            Abre_Comp_Indiv_Gar_1 = FALSE
            Fecha_Comp_Indiv_Gar_1 = TRUE

            Abre_Comp_Indiv_Gar_3 = FALSE
            Fecha_Comp_Indiv_Gar_3 = TRUE

            Abre_Comp_Indiv_Gar_4 = FALSE
            Fecha_Comp_Indiv_Gar_4 = TRUE

            Abre_Comp_Indiv_Gar_6 = FALSE
            Fecha_Comp_Indiv_Gar_6 = TRUE

            Ava_Cil_1_Gar_1 = TRUE
            Rec_Cil_1_Gar_1 = FALSE

            Ava_Cil_1_Gar_2 = TRUE
            Rec_Cil_1_Gar_2 = FALSE

            Ava_Cil_1_Gar_3 = TRUE
            Rec_Cil_1_Gar_3 = FALSE

            Ava_Cil_1_Gar_4 = TRUE
            Rec_Cil_1_Gar_4 = FALSE

            Ava_Cil_1_Gar_5 = TRUE
            Rec_Cil_1_Gar_5 = FALSE

            Ava_Cil_1_Gar_6 = TRUE
            Rec_Cil_1_Gar_6 = FALSE

            Ava_Cil_2_Gar_1 = TRUE
            Rec_Cil_2_Gar_1 = FALSE

            Ava_Cil_2_Gar_2 = TRUE
            Rec_Cil_2_Gar_2 = FALSE

            Ava_Cil_2_Gar_3 = TRUE
            Rec_Cil_2_Gar_3 = FALSE

            Ava_Cil_2_Gar_4 = TRUE
            Rec_Cil_2_Gar_4 = FALSE

            Ava_Cil_2_Gar_5 = TRUE
            Rec_Cil_2_Gar_5 = FALSE

            Ava_Cil_2_Gar_6 = TRUE
            Rec_Cil_2_Gar_6 = FALSE



         CASE 162
            Abre_Gar_Triplo_Lado_A = TRUE
            Fecha_Gar_Triplo_Lado_A = FALSE

            Abre_Gar_Triplo_Lado_B = TRUE
            Fecha_Gar_Triplo_Lado_B = FALSE

            Abre_Comp_Indiv_Gar_1 = FALSE
            Fecha_Comp_Indiv_Gar_1 = TRUE

            Abre_Comp_Indiv_Gar_3 = FALSE
            Fecha_Comp_Indiv_Gar_3 = TRUE

            Abre_Comp_Indiv_Gar_4 = FALSE
            Fecha_Comp_Indiv_Gar_4 = TRUE

            Abre_Comp_Indiv_Gar_6 = TRUE
            Fecha_Comp_Indiv_Gar_6 = FALSE

            Ava_Cil_1_Gar_1 = TRUE
            Rec_Cil_1_Gar_1 = FALSE

            Ava_Cil_1_Gar_2 = TRUE
            Rec_Cil_1_Gar_2 = FALSE

            Ava_Cil_1_Gar_3 = TRUE
            Rec_Cil_1_Gar_3 = FALSE

            Ava_Cil_1_Gar_4 = TRUE
            Rec_Cil_1_Gar_4 = FALSE

            Ava_Cil_1_Gar_5 = TRUE
            Rec_Cil_1_Gar_5 = FALSE

            Ava_Cil_1_Gar_6 = TRUE
            Rec_Cil_1_Gar_6 = FALSE

            Ava_Cil_2_Gar_1 = TRUE
            Rec_Cil_2_Gar_1 = FALSE

            Ava_Cil_2_Gar_2 = TRUE
            Rec_Cil_2_Gar_2 = FALSE

            Ava_Cil_2_Gar_3 = TRUE
            Rec_Cil_2_Gar_3 = FALSE

            Ava_Cil_2_Gar_4 = TRUE
            Rec_Cil_2_Gar_4 = FALSE

            Ava_Cil_2_Gar_5 = TRUE
            Rec_Cil_2_Gar_5 = FALSE

            Ava_Cil_2_Gar_6 = TRUE
            Rec_Cil_2_Gar_6 = FALSE

         CASE 61
            Abre_Gar_Triplo_Lado_A = TRUE
            Fecha_Gar_Triplo_Lado_A = FALSE

            Abre_Gar_Triplo_Lado_B = TRUE
            Fecha_Gar_Triplo_Lado_B = FALSE

            Abre_Comp_Indiv_Gar_1 = TRUE
            Fecha_Comp_Indiv_Gar_1 = FALSE

            Abre_Comp_Indiv_Gar_3 = FALSE
            Fecha_Comp_Indiv_Gar_3 = TRUE

            Abre_Comp_Indiv_Gar_4 = FALSE
            Fecha_Comp_Indiv_Gar_4 = TRUE

            Abre_Comp_Indiv_Gar_6 = TRUE
            Fecha_Comp_Indiv_Gar_6 = FALSE

            Ava_Cil_1_Gar_1 = TRUE
            Rec_Cil_1_Gar_1 = FALSE

            Ava_Cil_1_Gar_2 = TRUE
            Rec_Cil_1_Gar_2 = FALSE

            Ava_Cil_1_Gar_3 = TRUE
            Rec_Cil_1_Gar_3 = FALSE

            Ava_Cil_1_Gar_4 = TRUE
            Rec_Cil_1_Gar_4 = FALSE

            Ava_Cil_1_Gar_5 = TRUE
            Rec_Cil_1_Gar_5 = FALSE

            Ava_Cil_1_Gar_6 = TRUE
            Rec_Cil_1_Gar_6 = FALSE

            Ava_Cil_2_Gar_1 = TRUE
            Rec_Cil_2_Gar_1 = FALSE

            Ava_Cil_2_Gar_2 = TRUE
            Rec_Cil_2_Gar_2 = FALSE

            Ava_Cil_2_Gar_3 = TRUE
            Rec_Cil_2_Gar_3 = FALSE

            Ava_Cil_2_Gar_4 = TRUE
            Rec_Cil_2_Gar_4 = FALSE

            Ava_Cil_2_Gar_5 = TRUE
            Rec_Cil_2_Gar_5 = FALSE

            Ava_Cil_2_Gar_6 = TRUE
            Rec_Cil_2_Gar_6 = FALSE


         CASE 62
            Abre_Gar_Triplo_Lado_A = TRUE
            Fecha_Gar_Triplo_Lado_A = FALSE

            Abre_Gar_Triplo_Lado_B = TRUE
            Fecha_Gar_Triplo_Lado_B = FALSE

            Abre_Comp_Indiv_Gar_1 = TRUE
            Fecha_Comp_Indiv_Gar_1 = FALSE

            Abre_Comp_Indiv_Gar_3 = FALSE
            Fecha_Comp_Indiv_Gar_3 = TRUE

            Abre_Comp_Indiv_Gar_4 = FALSE
            Fecha_Comp_Indiv_Gar_4 = TRUE

            Abre_Comp_Indiv_Gar_6 = TRUE
            Fecha_Comp_Indiv_Gar_6 = FALSE

            Ava_Cil_1_Gar_1 = TRUE
            Rec_Cil_1_Gar_1 = FALSE

            Ava_Cil_1_Gar_2 = TRUE
            Rec_Cil_1_Gar_2 = FALSE

            Ava_Cil_1_Gar_3 = TRUE
            Rec_Cil_1_Gar_3 = FALSE

            Ava_Cil_1_Gar_4 = TRUE
            Rec_Cil_1_Gar_4 = FALSE

            Ava_Cil_1_Gar_5 = TRUE
            Rec_Cil_1_Gar_5 = FALSE

            Ava_Cil_1_Gar_6 = TRUE
            Rec_Cil_1_Gar_6 = FALSE

            Ava_Cil_2_Gar_1 = TRUE
            Rec_Cil_2_Gar_1 = FALSE

            Ava_Cil_2_Gar_2 = TRUE
            Rec_Cil_2_Gar_2 = FALSE

            Ava_Cil_2_Gar_3 = TRUE
            Rec_Cil_2_Gar_3 = FALSE

            Ava_Cil_2_Gar_4 = TRUE
            Rec_Cil_2_Gar_4 = FALSE

            Ava_Cil_2_Gar_5 = TRUE
            Rec_Cil_2_Gar_5 = FALSE

            Ava_Cil_2_Gar_6 = TRUE
            Rec_Cil_2_Gar_6 = FALSE

         CASE 191
            Abre_Gar_Triplo_Lado_A = TRUE
            Fecha_Gar_Triplo_Lado_A = FALSE

            Abre_Gar_Triplo_Lado_B = TRUE
            Fecha_Gar_Triplo_Lado_B = FALSE

            Abre_Comp_Indiv_Gar_1 = FALSE
            Fecha_Comp_Indiv_Gar_1 = TRUE

            Abre_Comp_Indiv_Gar_3 = FALSE
            Fecha_Comp_Indiv_Gar_3 = TRUE

            Abre_Comp_Indiv_Gar_4 = FALSE
            Fecha_Comp_Indiv_Gar_4 = TRUE

            Abre_Comp_Indiv_Gar_6 = FALSE
            Fecha_Comp_Indiv_Gar_6 = TRUE

            Ava_Cil_1_Gar_1 = TRUE
            Rec_Cil_1_Gar_1 = FALSE

            Ava_Cil_1_Gar_2 = TRUE
            Rec_Cil_1_Gar_2 = FALSE

            Ava_Cil_1_Gar_3 = TRUE
            Rec_Cil_1_Gar_3 = FALSE

            Ava_Cil_1_Gar_4 = TRUE
            Rec_Cil_1_Gar_4 = FALSE

            Ava_Cil_1_Gar_5 = TRUE
            Rec_Cil_1_Gar_5 = FALSE

            Ava_Cil_1_Gar_6 = TRUE
            Rec_Cil_1_Gar_6 = FALSE

            Ava_Cil_2_Gar_1 = TRUE
            Rec_Cil_2_Gar_1 = FALSE

            Ava_Cil_2_Gar_2 = TRUE
            Rec_Cil_2_Gar_2 = FALSE

            Ava_Cil_2_Gar_3 = TRUE
            Rec_Cil_2_Gar_3 = FALSE

            Ava_Cil_2_Gar_4 = TRUE
            Rec_Cil_2_Gar_4 = FALSE

            Ava_Cil_2_Gar_5 = TRUE
            Rec_Cil_2_Gar_5 = FALSE

            Ava_Cil_2_Gar_6 = TRUE
            Rec_Cil_2_Gar_6 = FALSE

         CASE 192
            Abre_Gar_Triplo_Lado_A = TRUE
            Fecha_Gar_Triplo_Lado_A = FALSE

            Abre_Gar_Triplo_Lado_B = TRUE
            Fecha_Gar_Triplo_Lado_B = FALSE

            Abre_Comp_Indiv_Gar_1 = FALSE
            Fecha_Comp_Indiv_Gar_1 = TRUE

            Abre_Comp_Indiv_Gar_3 = FALSE
            Fecha_Comp_Indiv_Gar_3 = TRUE

            Abre_Comp_Indiv_Gar_4 = FALSE
            Fecha_Comp_Indiv_Gar_4 = TRUE

            Abre_Comp_Indiv_Gar_6 = FALSE
            Fecha_Comp_Indiv_Gar_6 = TRUE

            Ava_Cil_1_Gar_1 = TRUE
            Rec_Cil_1_Gar_1 = FALSE

            Ava_Cil_1_Gar_2 = TRUE
            Rec_Cil_1_Gar_2 = FALSE

            Ava_Cil_1_Gar_3 = TRUE
            Rec_Cil_1_Gar_3 = FALSE

            Ava_Cil_1_Gar_4 = TRUE
            Rec_Cil_1_Gar_4 = FALSE

            Ava_Cil_1_Gar_5 = TRUE
            Rec_Cil_1_Gar_5 = FALSE

            Ava_Cil_1_Gar_6 = TRUE
            Rec_Cil_1_Gar_6 = FALSE

            Ava_Cil_2_Gar_1 = TRUE
            Rec_Cil_2_Gar_1 = FALSE

            Ava_Cil_2_Gar_2 = TRUE
            Rec_Cil_2_Gar_2 = FALSE

            Ava_Cil_2_Gar_3 = TRUE
            Rec_Cil_2_Gar_3 = FALSE

            Ava_Cil_2_Gar_4 = TRUE
            Rec_Cil_2_Gar_4 = FALSE

            Ava_Cil_2_Gar_5 = TRUE
            Rec_Cil_2_Gar_5 = FALSE

            Ava_Cil_2_Gar_6 = TRUE
            Rec_Cil_2_Gar_6 = FALSE

         CASE 81
            Abre_Gar_Triplo_Lado_A = TRUE
            Fecha_Gar_Triplo_Lado_A = FALSE

            Abre_Gar_Triplo_Lado_B = TRUE
            Fecha_Gar_Triplo_Lado_B = FALSE

            Abre_Comp_Indiv_Gar_1 = FALSE
            Fecha_Comp_Indiv_Gar_1 = TRUE

            Abre_Comp_Indiv_Gar_3 = FALSE
            Fecha_Comp_Indiv_Gar_3 = TRUE

            Abre_Comp_Indiv_Gar_4 = FALSE
            Fecha_Comp_Indiv_Gar_4 = TRUE

            Abre_Comp_Indiv_Gar_6 = TRUE
            Fecha_Comp_Indiv_Gar_6 = FALSE

            Ava_Cil_1_Gar_1 = TRUE
            Rec_Cil_1_Gar_1 = FALSE

            Ava_Cil_1_Gar_2 = TRUE
            Rec_Cil_1_Gar_2 = FALSE

            Ava_Cil_1_Gar_3 = TRUE
            Rec_Cil_1_Gar_3 = FALSE

            Ava_Cil_1_Gar_4 = TRUE
            Rec_Cil_1_Gar_4 = FALSE

            Ava_Cil_1_Gar_5 = TRUE
            Rec_Cil_1_Gar_5 = FALSE

            Ava_Cil_1_Gar_6 = TRUE
            Rec_Cil_1_Gar_6 = FALSE

            Ava_Cil_2_Gar_1 = TRUE
            Rec_Cil_2_Gar_1 = FALSE

            Ava_Cil_2_Gar_2 = TRUE
            Rec_Cil_2_Gar_2 = FALSE

            Ava_Cil_2_Gar_3 = TRUE
            Rec_Cil_2_Gar_3 = FALSE

            Ava_Cil_2_Gar_4 = TRUE
            Rec_Cil_2_Gar_4 = FALSE

            Ava_Cil_2_Gar_5 = TRUE
            Rec_Cil_2_Gar_5 = FALSE

            Ava_Cil_2_Gar_6 = TRUE
            Rec_Cil_2_Gar_6 = FALSE

         CASE 82
            Abre_Gar_Triplo_Lado_A = TRUE
            Fecha_Gar_Triplo_Lado_A = FALSE

            Abre_Gar_Triplo_Lado_B = TRUE
            Fecha_Gar_Triplo_Lado_B = FALSE

            Abre_Comp_Indiv_Gar_1 = FALSE
            Fecha_Comp_Indiv_Gar_1 = TRUE

            Abre_Comp_Indiv_Gar_3 = TRUE
            Fecha_Comp_Indiv_Gar_3 = FALSE

            Abre_Comp_Indiv_Gar_4 = TRUE
            Fecha_Comp_Indiv_Gar_4 = FALSE

            Abre_Comp_Indiv_Gar_6 = FALSE
            Fecha_Comp_Indiv_Gar_6 = TRUE

            Ava_Cil_1_Gar_1 = TRUE
            Rec_Cil_1_Gar_1 = FALSE

            Ava_Cil_1_Gar_2 = TRUE
            Rec_Cil_1_Gar_2 = FALSE

            Ava_Cil_1_Gar_3 = TRUE
            Rec_Cil_1_Gar_3 = FALSE

            Ava_Cil_1_Gar_4 = TRUE
            Rec_Cil_1_Gar_4 = FALSE

            Ava_Cil_1_Gar_5 = TRUE
            Rec_Cil_1_Gar_5 = FALSE

            Ava_Cil_1_Gar_6 = TRUE
            Rec_Cil_1_Gar_6 = FALSE

            Ava_Cil_2_Gar_1 = TRUE
            Rec_Cil_2_Gar_1 = FALSE

            Ava_Cil_2_Gar_2 = TRUE
            Rec_Cil_2_Gar_2 = FALSE

            Ava_Cil_2_Gar_3 = TRUE
            Rec_Cil_2_Gar_3 = FALSE

            Ava_Cil_2_Gar_4 = TRUE
            Rec_Cil_2_Gar_4 = FALSE

            Ava_Cil_2_Gar_5 = TRUE
            Rec_Cil_2_Gar_5 = FALSE

            Ava_Cil_2_Gar_6 = TRUE
            Rec_Cil_2_Gar_6 = FALSE

         CASE 91
            Abre_Gar_Triplo_Lado_A = TRUE
            Fecha_Gar_Triplo_Lado_A = FALSE

            Abre_Gar_Triplo_Lado_B = TRUE
            Fecha_Gar_Triplo_Lado_B = FALSE

            Abre_Comp_Indiv_Gar_1 = FALSE
            Fecha_Comp_Indiv_Gar_1 = TRUE

            Abre_Comp_Indiv_Gar_3 = TRUE
            Fecha_Comp_Indiv_Gar_3 = FALSE

            Abre_Comp_Indiv_Gar_4 = TRUE
            Fecha_Comp_Indiv_Gar_4 = FALSE

            Abre_Comp_Indiv_Gar_6 = FALSE
            Fecha_Comp_Indiv_Gar_6 = TRUE

            Ava_Cil_1_Gar_1 = TRUE
            Rec_Cil_1_Gar_1 = FALSE

            Ava_Cil_1_Gar_2 = TRUE
            Rec_Cil_1_Gar_2 = FALSE

            Ava_Cil_1_Gar_3 = TRUE
            Rec_Cil_1_Gar_3 = FALSE

            Ava_Cil_1_Gar_4 = TRUE
            Rec_Cil_1_Gar_4 = FALSE

            Ava_Cil_1_Gar_5 = TRUE
            Rec_Cil_1_Gar_5 = FALSE

            Ava_Cil_1_Gar_6 = TRUE
            Rec_Cil_1_Gar_6 = FALSE

            Ava_Cil_2_Gar_1 = TRUE
            Rec_Cil_2_Gar_1 = FALSE

            Ava_Cil_2_Gar_2 = TRUE
            Rec_Cil_2_Gar_2 = FALSE

            Ava_Cil_2_Gar_3 = TRUE
            Rec_Cil_2_Gar_3 = FALSE

            Ava_Cil_2_Gar_4 = TRUE
            Rec_Cil_2_Gar_4 = FALSE

            Ava_Cil_2_Gar_5 = TRUE
            Rec_Cil_2_Gar_5 = FALSE

            Ava_Cil_2_Gar_6 = TRUE
            Rec_Cil_2_Gar_6 = FALSE


         CASE 92
            Abre_Gar_Triplo_Lado_A = TRUE
            Fecha_Gar_Triplo_Lado_A = FALSE

            Abre_Gar_Triplo_Lado_B = TRUE
            Fecha_Gar_Triplo_Lado_B = FALSE

            Abre_Comp_Indiv_Gar_1 = FALSE
            Fecha_Comp_Indiv_Gar_1 = TRUE

            Abre_Comp_Indiv_Gar_3 = FALSE
            Fecha_Comp_Indiv_Gar_3 = TRUE

            Abre_Comp_Indiv_Gar_4 = FALSE
            Fecha_Comp_Indiv_Gar_4 = TRUE

            Abre_Comp_Indiv_Gar_6 = TRUE
            Fecha_Comp_Indiv_Gar_6 = FALSE

            Ava_Cil_1_Gar_1 = TRUE
            Rec_Cil_1_Gar_1 = FALSE

            Ava_Cil_1_Gar_2 = TRUE
            Rec_Cil_1_Gar_2 = FALSE

            Ava_Cil_1_Gar_3 = TRUE
            Rec_Cil_1_Gar_3 = FALSE

            Ava_Cil_1_Gar_4 = TRUE
            Rec_Cil_1_Gar_4 = FALSE

            Ava_Cil_1_Gar_5 = TRUE
            Rec_Cil_1_Gar_5 = FALSE

            Ava_Cil_1_Gar_6 = TRUE
            Rec_Cil_1_Gar_6 = FALSE

            Ava_Cil_2_Gar_1 = TRUE
            Rec_Cil_2_Gar_1 = FALSE

            Ava_Cil_2_Gar_2 = TRUE
            Rec_Cil_2_Gar_2 = FALSE

            Ava_Cil_2_Gar_3 = TRUE
            Rec_Cil_2_Gar_3 = FALSE

            Ava_Cil_2_Gar_4 = TRUE
            Rec_Cil_2_Gar_4 = FALSE

            Ava_Cil_2_Gar_5 = TRUE
            Rec_Cil_2_Gar_5 = FALSE

            Ava_Cil_2_Gar_6 = TRUE
            Rec_Cil_2_Gar_6 = FALSE

         CASE 151
            Abre_Gar_Triplo_Lado_A = TRUE
            Fecha_Gar_Triplo_Lado_A = FALSE

            Abre_Gar_Triplo_Lado_B = TRUE
            Fecha_Gar_Triplo_Lado_B = FALSE

            Abre_Comp_Indiv_Gar_1 = TRUE
            Fecha_Comp_Indiv_Gar_1 = FALSE

            Abre_Comp_Indiv_Gar_3 = FALSE
            Fecha_Comp_Indiv_Gar_3 = TRUE

            Abre_Comp_Indiv_Gar_4 = FALSE
            Fecha_Comp_Indiv_Gar_4 = TRUE

            Abre_Comp_Indiv_Gar_6 = TRUE
            Fecha_Comp_Indiv_Gar_6 = FALSE

            Ava_Cil_1_Gar_1 = TRUE
            Rec_Cil_1_Gar_1 = FALSE

            Ava_Cil_1_Gar_2 = TRUE
            Rec_Cil_1_Gar_2 = FALSE

            Ava_Cil_1_Gar_3 = TRUE
            Rec_Cil_1_Gar_3 = FALSE

            Ava_Cil_1_Gar_4 = TRUE
            Rec_Cil_1_Gar_4 = FALSE

            Ava_Cil_1_Gar_5 = TRUE
            Rec_Cil_1_Gar_5 = FALSE

            Ava_Cil_1_Gar_6 = TRUE
            Rec_Cil_1_Gar_6 = FALSE

            Ava_Cil_2_Gar_1 = TRUE
            Rec_Cil_2_Gar_1 = FALSE

            Ava_Cil_2_Gar_2 = TRUE
            Rec_Cil_2_Gar_2 = FALSE

            Ava_Cil_2_Gar_3 = TRUE
            Rec_Cil_2_Gar_3 = FALSE

            Ava_Cil_2_Gar_4 = TRUE
            Rec_Cil_2_Gar_4 = FALSE

            Ava_Cil_2_Gar_5 = TRUE
            Rec_Cil_2_Gar_5 = FALSE

            Ava_Cil_2_Gar_6 = TRUE
            Rec_Cil_2_Gar_6 = FALSE

         CASE 141
            Abre_Gar_Triplo_Lado_A = TRUE
            Fecha_Gar_Triplo_Lado_A = FALSE

            Abre_Gar_Triplo_Lado_B = TRUE
            Fecha_Gar_Triplo_Lado_B = FALSE

            Abre_Comp_Indiv_Gar_1 = FALSE
            Fecha_Comp_Indiv_Gar_1 = TRUE

            Abre_Comp_Indiv_Gar_3 = FALSE
            Fecha_Comp_Indiv_Gar_3 = TRUE

            Abre_Comp_Indiv_Gar_4 = FALSE
            Fecha_Comp_Indiv_Gar_4 = TRUE

            Abre_Comp_Indiv_Gar_6 = FALSE
            Fecha_Comp_Indiv_Gar_6 = TRUE

            Ava_Cil_1_Gar_1 = TRUE
            Rec_Cil_1_Gar_1 = FALSE

            Ava_Cil_1_Gar_2 = TRUE
            Rec_Cil_1_Gar_2 = FALSE

            Ava_Cil_1_Gar_3 = TRUE
            Rec_Cil_1_Gar_3 = FALSE

            Ava_Cil_1_Gar_4 = TRUE
            Rec_Cil_1_Gar_4 = FALSE

            Ava_Cil_1_Gar_5 = TRUE
            Rec_Cil_1_Gar_5 = FALSE

            Ava_Cil_1_Gar_6 = TRUE
            Rec_Cil_1_Gar_6 = FALSE

            Ava_Cil_2_Gar_1 = TRUE
            Rec_Cil_2_Gar_1 = FALSE

            Ava_Cil_2_Gar_2 = TRUE
            Rec_Cil_2_Gar_2 = FALSE

            Ava_Cil_2_Gar_3 = TRUE
            Rec_Cil_2_Gar_3 = FALSE

            Ava_Cil_2_Gar_4 = TRUE
            Rec_Cil_2_Gar_4 = FALSE

            Ava_Cil_2_Gar_5 = TRUE
            Rec_Cil_2_Gar_5 = FALSE

            Ava_Cil_2_Gar_6 = TRUE
            Rec_Cil_2_Gar_6 = FALSE

         CASE 142
            Abre_Gar_Triplo_Lado_A = TRUE
            Fecha_Gar_Triplo_Lado_A = FALSE

            Abre_Gar_Triplo_Lado_B = TRUE
            Fecha_Gar_Triplo_Lado_B = FALSE

            Abre_Comp_Indiv_Gar_1 = FALSE
            Fecha_Comp_Indiv_Gar_1 = TRUE

            Abre_Comp_Indiv_Gar_3 = FALSE
            Fecha_Comp_Indiv_Gar_3 = TRUE

            Abre_Comp_Indiv_Gar_4 = FALSE
            Fecha_Comp_Indiv_Gar_4 = TRUE

            Abre_Comp_Indiv_Gar_6 = FALSE
            Fecha_Comp_Indiv_Gar_6 = TRUE

            Ava_Cil_1_Gar_1 = TRUE
            Rec_Cil_1_Gar_1 = FALSE

            Ava_Cil_1_Gar_2 = TRUE
            Rec_Cil_1_Gar_2 = FALSE

            Ava_Cil_1_Gar_3 = TRUE
            Rec_Cil_1_Gar_3 = FALSE

            Ava_Cil_1_Gar_4 = TRUE
            Rec_Cil_1_Gar_4 = FALSE

            Ava_Cil_1_Gar_5 = TRUE
            Rec_Cil_1_Gar_5 = FALSE

            Ava_Cil_1_Gar_6 = TRUE
            Rec_Cil_1_Gar_6 = FALSE

            Ava_Cil_2_Gar_1 = TRUE
            Rec_Cil_2_Gar_1 = FALSE

            Ava_Cil_2_Gar_2 = TRUE
            Rec_Cil_2_Gar_2 = FALSE

            Ava_Cil_2_Gar_3 = TRUE
            Rec_Cil_2_Gar_3 = FALSE

            Ava_Cil_2_Gar_4 = TRUE
            Rec_Cil_2_Gar_4 = FALSE

            Ava_Cil_2_Gar_5 = TRUE
            Rec_Cil_2_Gar_5 = FALSE

            Ava_Cil_2_Gar_6 = TRUE
            Rec_Cil_2_Gar_6 = FALSE

         CASE 171
            Abre_Gar_Triplo_Lado_A = TRUE
            Fecha_Gar_Triplo_Lado_A = FALSE

            Abre_Gar_Triplo_Lado_B = TRUE
            Fecha_Gar_Triplo_Lado_B = FALSE

            Abre_Comp_Indiv_Gar_1 = TRUE
            Fecha_Comp_Indiv_Gar_1 = FALSE

            Abre_Comp_Indiv_Gar_3 = FALSE
            Fecha_Comp_Indiv_Gar_3 = TRUE

            Abre_Comp_Indiv_Gar_4 = FALSE
            Fecha_Comp_Indiv_Gar_4 = TRUE

            Abre_Comp_Indiv_Gar_6 = FALSE
            Fecha_Comp_Indiv_Gar_6 = TRUE

            Ava_Cil_1_Gar_1 = TRUE
            Rec_Cil_1_Gar_1 = FALSE

            Ava_Cil_1_Gar_2 = TRUE
            Rec_Cil_1_Gar_2 = FALSE

            Ava_Cil_1_Gar_3 = TRUE
            Rec_Cil_1_Gar_3 = FALSE

            Ava_Cil_1_Gar_4 = TRUE
            Rec_Cil_1_Gar_4 = FALSE

            Ava_Cil_1_Gar_5 = TRUE
            Rec_Cil_1_Gar_5 = FALSE

            Ava_Cil_1_Gar_6 = TRUE
            Rec_Cil_1_Gar_6 = FALSE

            Ava_Cil_2_Gar_1 = TRUE
            Rec_Cil_2_Gar_1 = FALSE

            Ava_Cil_2_Gar_2 = TRUE
            Rec_Cil_2_Gar_2 = FALSE

            Ava_Cil_2_Gar_3 = TRUE
            Rec_Cil_2_Gar_3 = FALSE

            Ava_Cil_2_Gar_4 = TRUE
            Rec_Cil_2_Gar_4 = FALSE

            Ava_Cil_2_Gar_5 = TRUE
            Rec_Cil_2_Gar_5 = FALSE

            Ava_Cil_2_Gar_6 = TRUE
            Rec_Cil_2_Gar_6 = FALSE


         CASE 172
            Abre_Gar_Triplo_Lado_A = TRUE
            Fecha_Gar_Triplo_Lado_A = FALSE

            Abre_Gar_Triplo_Lado_B = TRUE
            Fecha_Gar_Triplo_Lado_B = FALSE

            Abre_Comp_Indiv_Gar_1 = TRUE
            Fecha_Comp_Indiv_Gar_1 = FALSE

            Abre_Comp_Indiv_Gar_3 = FALSE
            Fecha_Comp_Indiv_Gar_3 = TRUE

            Abre_Comp_Indiv_Gar_4 = FALSE
            Fecha_Comp_Indiv_Gar_4 = TRUE

            Abre_Comp_Indiv_Gar_6 = TRUE
            Fecha_Comp_Indiv_Gar_6 = FALSE

            Ava_Cil_1_Gar_1 = TRUE
            Rec_Cil_1_Gar_1 = FALSE

            Ava_Cil_1_Gar_2 = TRUE
            Rec_Cil_1_Gar_2 = FALSE

            Ava_Cil_1_Gar_3 = TRUE
            Rec_Cil_1_Gar_3 = FALSE

            Ava_Cil_1_Gar_4 = TRUE
            Rec_Cil_1_Gar_4 = FALSE

            Ava_Cil_1_Gar_5 = TRUE
            Rec_Cil_1_Gar_5 = FALSE

            Ava_Cil_1_Gar_6 = TRUE
            Rec_Cil_1_Gar_6 = FALSE

            Ava_Cil_2_Gar_1 = TRUE
            Rec_Cil_2_Gar_1 = FALSE

            Ava_Cil_2_Gar_2 = TRUE
            Rec_Cil_2_Gar_2 = FALSE

            Ava_Cil_2_Gar_3 = TRUE
            Rec_Cil_2_Gar_3 = FALSE

            Ava_Cil_2_Gar_4 = TRUE
            Rec_Cil_2_Gar_4 = FALSE

            Ava_Cil_2_Gar_5 = TRUE
            Rec_Cil_2_Gar_5 = FALSE

            Ava_Cil_2_Gar_6 = TRUE
            Rec_Cil_2_Gar_6 = FALSE

         CASE 173
            Abre_Gar_Triplo_Lado_A = TRUE
            Fecha_Gar_Triplo_Lado_A = FALSE

            Abre_Gar_Triplo_Lado_B = TRUE
            Fecha_Gar_Triplo_Lado_B = FALSE

            Abre_Comp_Indiv_Gar_1 = TRUE
            Fecha_Comp_Indiv_Gar_1 = FALSE

            Abre_Comp_Indiv_Gar_3 = FALSE
            Fecha_Comp_Indiv_Gar_3 = TRUE

            Abre_Comp_Indiv_Gar_4 = FALSE
            Fecha_Comp_Indiv_Gar_4 = TRUE

            Abre_Comp_Indiv_Gar_6 = TRUE
            Fecha_Comp_Indiv_Gar_6 = FALSE

            Ava_Cil_1_Gar_1 = TRUE
            Rec_Cil_1_Gar_1 = FALSE

            Ava_Cil_1_Gar_2 = TRUE
            Rec_Cil_1_Gar_2 = FALSE

            Ava_Cil_1_Gar_3 = TRUE
            Rec_Cil_1_Gar_3 = FALSE

            Ava_Cil_1_Gar_4 = TRUE
            Rec_Cil_1_Gar_4 = FALSE

            Ava_Cil_1_Gar_5 = TRUE
            Rec_Cil_1_Gar_5 = FALSE

            Ava_Cil_1_Gar_6 = TRUE
            Rec_Cil_1_Gar_6 = FALSE

            Ava_Cil_2_Gar_1 = TRUE
            Rec_Cil_2_Gar_1 = FALSE

            Ava_Cil_2_Gar_2 = TRUE
            Rec_Cil_2_Gar_2 = FALSE

            Ava_Cil_2_Gar_3 = TRUE
            Rec_Cil_2_Gar_3 = FALSE

            Ava_Cil_2_Gar_4 = TRUE
            Rec_Cil_2_Gar_4 = FALSE

            Ava_Cil_2_Gar_5 = TRUE
            Rec_Cil_2_Gar_5 = FALSE

            Ava_Cil_2_Gar_6 = TRUE
            Rec_Cil_2_Gar_6 = FALSE


         CASE 71
            Abre_Gar_Triplo_Lado_A = TRUE
            Fecha_Gar_Triplo_Lado_A = FALSE

            Abre_Gar_Triplo_Lado_B = TRUE
            Fecha_Gar_Triplo_Lado_B = FALSE

            Abre_Comp_Indiv_Gar_1 = FALSE
            Fecha_Comp_Indiv_Gar_1 = TRUE

            Abre_Comp_Indiv_Gar_3 = TRUE
            Fecha_Comp_Indiv_Gar_3 = FALSE

            Abre_Comp_Indiv_Gar_4 = TRUE
            Fecha_Comp_Indiv_Gar_4 = FALSE

            Abre_Comp_Indiv_Gar_6 = FALSE
            Fecha_Comp_Indiv_Gar_6 = TRUE

            Ava_Cil_1_Gar_1 = TRUE
            Rec_Cil_1_Gar_1 = FALSE

            Ava_Cil_1_Gar_2 = TRUE
            Rec_Cil_1_Gar_2 = FALSE

            Ava_Cil_1_Gar_3 = TRUE
            Rec_Cil_1_Gar_3 = FALSE

            Ava_Cil_1_Gar_4 = TRUE
            Rec_Cil_1_Gar_4 = FALSE

            Ava_Cil_1_Gar_5 = TRUE
            Rec_Cil_1_Gar_5 = FALSE

            Ava_Cil_1_Gar_6 = TRUE
            Rec_Cil_1_Gar_6 = FALSE

            Ava_Cil_2_Gar_1 = TRUE
            Rec_Cil_2_Gar_1 = FALSE

            Ava_Cil_2_Gar_2 = TRUE
            Rec_Cil_2_Gar_2 = FALSE

            Ava_Cil_2_Gar_3 = TRUE
            Rec_Cil_2_Gar_3 = FALSE

            Ava_Cil_2_Gar_4 = TRUE
            Rec_Cil_2_Gar_4 = FALSE

            Ava_Cil_2_Gar_5 = TRUE
            Rec_Cil_2_Gar_5 = FALSE

            Ava_Cil_2_Gar_6 = TRUE
            Rec_Cil_2_Gar_6 = FALSE


         CASE 72
            Abre_Gar_Triplo_Lado_A = TRUE
            Fecha_Gar_Triplo_Lado_A = FALSE

            Abre_Gar_Triplo_Lado_B = TRUE
            Fecha_Gar_Triplo_Lado_B = FALSE

            Abre_Comp_Indiv_Gar_1 = TRUE
            Fecha_Comp_Indiv_Gar_1 = FALSE

            Abre_Comp_Indiv_Gar_3 = FALSE
            Fecha_Comp_Indiv_Gar_3 = TRUE

            Abre_Comp_Indiv_Gar_4 = TRUE
            Fecha_Comp_Indiv_Gar_4 = FALSE

            Abre_Comp_Indiv_Gar_6 = FALSE
            Fecha_Comp_Indiv_Gar_6 = TRUE

            Ava_Cil_1_Gar_1 = TRUE
            Rec_Cil_1_Gar_1 = FALSE

            Ava_Cil_1_Gar_2 = TRUE
            Rec_Cil_1_Gar_2 = FALSE

            Ava_Cil_1_Gar_3 = TRUE
            Rec_Cil_1_Gar_3 = FALSE

            Ava_Cil_1_Gar_4 = TRUE
            Rec_Cil_1_Gar_4 = FALSE

            Ava_Cil_1_Gar_5 = TRUE
            Rec_Cil_1_Gar_5 = FALSE

            Ava_Cil_1_Gar_6 = TRUE
            Rec_Cil_1_Gar_6 = FALSE

            Ava_Cil_2_Gar_1 = TRUE
            Rec_Cil_2_Gar_1 = FALSE

            Ava_Cil_2_Gar_2 = TRUE
            Rec_Cil_2_Gar_2 = FALSE

            Ava_Cil_2_Gar_3 = TRUE
            Rec_Cil_2_Gar_3 = FALSE

            Ava_Cil_2_Gar_4 = TRUE
            Rec_Cil_2_Gar_4 = FALSE

            Ava_Cil_2_Gar_5 = TRUE
            Rec_Cil_2_Gar_5 = FALSE

            Ava_Cil_2_Gar_6 = TRUE
            Rec_Cil_2_Gar_6 = FALSE


         CASE 73
            Abre_Gar_Triplo_Lado_A = TRUE
            Fecha_Gar_Triplo_Lado_A = FALSE

            Abre_Gar_Triplo_Lado_B = TRUE
            Fecha_Gar_Triplo_Lado_B = FALSE

            Abre_Comp_Indiv_Gar_1 = TRUE
            Fecha_Comp_Indiv_Gar_1 = FALSE

            Abre_Comp_Indiv_Gar_3 = TRUE
            Fecha_Comp_Indiv_Gar_3 = FALSE

            Abre_Comp_Indiv_Gar_4 = TRUE
            Fecha_Comp_Indiv_Gar_4 = FALSE

            Abre_Comp_Indiv_Gar_6 = TRUE
            Fecha_Comp_Indiv_Gar_6 = FALSE

            Ava_Cil_1_Gar_1 = TRUE
            Rec_Cil_1_Gar_1 = FALSE

            Ava_Cil_1_Gar_2 = TRUE
            Rec_Cil_1_Gar_2 = FALSE

            Ava_Cil_1_Gar_3 = TRUE
            Rec_Cil_1_Gar_3 = FALSE

            Ava_Cil_1_Gar_4 = TRUE
            Rec_Cil_1_Gar_4 = FALSE

            Ava_Cil_1_Gar_5 = TRUE
            Rec_Cil_1_Gar_5 = FALSE

            Ava_Cil_1_Gar_6 = TRUE
            Rec_Cil_1_Gar_6 = FALSE

            Ava_Cil_2_Gar_1 = TRUE
            Rec_Cil_2_Gar_1 = FALSE

            Ava_Cil_2_Gar_2 = TRUE
            Rec_Cil_2_Gar_2 = FALSE

            Ava_Cil_2_Gar_3 = TRUE
            Rec_Cil_2_Gar_3 = FALSE

            Ava_Cil_2_Gar_4 = TRUE
            Rec_Cil_2_Gar_4 = FALSE

            Ava_Cil_2_Gar_5 = TRUE
            Rec_Cil_2_Gar_5 = FALSE

            Ava_Cil_2_Gar_6 = TRUE
            Rec_Cil_2_Gar_6 = FALSE


         CASE 51
            Abre_Gar_Triplo_Lado_A = TRUE
            Fecha_Gar_Triplo_Lado_A = FALSE

            Abre_Gar_Triplo_Lado_B = TRUE
            Fecha_Gar_Triplo_Lado_B = FALSE

            Abre_Comp_Indiv_Gar_1 = TRUE
            Fecha_Comp_Indiv_Gar_1 = FALSE

            Abre_Comp_Indiv_Gar_3 = TRUE
            Fecha_Comp_Indiv_Gar_3 = FALSE

            Abre_Comp_Indiv_Gar_4 = TRUE
            Fecha_Comp_Indiv_Gar_4 = FALSE

            Abre_Comp_Indiv_Gar_6 = TRUE
            Fecha_Comp_Indiv_Gar_6 = FALSE

            Ava_Cil_1_Gar_1 = TRUE
            Rec_Cil_1_Gar_1 = FALSE

            Ava_Cil_1_Gar_2 = TRUE
            Rec_Cil_1_Gar_2 = FALSE

            Ava_Cil_1_Gar_3 = TRUE
            Rec_Cil_1_Gar_3 = FALSE

            Ava_Cil_1_Gar_4 = TRUE
            Rec_Cil_1_Gar_4 = FALSE

            Ava_Cil_1_Gar_5 = TRUE
            Rec_Cil_1_Gar_5 = FALSE

            Ava_Cil_1_Gar_6 = TRUE
            Rec_Cil_1_Gar_6 = FALSE

            Ava_Cil_2_Gar_1 = TRUE
            Rec_Cil_2_Gar_1 = FALSE

            Ava_Cil_2_Gar_2 = TRUE
            Rec_Cil_2_Gar_2 = FALSE

            Ava_Cil_2_Gar_3 = TRUE
            Rec_Cil_2_Gar_3 = FALSE

            Ava_Cil_2_Gar_4 = TRUE
            Rec_Cil_2_Gar_4 = FALSE

            Ava_Cil_2_Gar_5 = TRUE
            Rec_Cil_2_Gar_5 = FALSE

            Ava_Cil_2_Gar_6 = TRUE
            Rec_Cil_2_Gar_6 = FALSE

         CASE 131
            Abre_Gar_Triplo_Lado_A = TRUE
            Fecha_Gar_Triplo_Lado_A = FALSE

            Abre_Gar_Triplo_Lado_B = TRUE
            Fecha_Gar_Triplo_Lado_B = FALSE

            Abre_Comp_Indiv_Gar_1 = TRUE
            Fecha_Comp_Indiv_Gar_1 = FALSE

            Abre_Comp_Indiv_Gar_3 = TRUE
            Fecha_Comp_Indiv_Gar_3 = FALSE

            Abre_Comp_Indiv_Gar_4 = TRUE
            Fecha_Comp_Indiv_Gar_4 = FALSE

            Abre_Comp_Indiv_Gar_6 = TRUE
            Fecha_Comp_Indiv_Gar_6 = FALSE

            Ava_Cil_1_Gar_1 = TRUE
            Rec_Cil_1_Gar_1 = FALSE

            Ava_Cil_1_Gar_2 = TRUE
            Rec_Cil_1_Gar_2 = FALSE

            Ava_Cil_1_Gar_3 = TRUE
            Rec_Cil_1_Gar_3 = FALSE

            Ava_Cil_1_Gar_4 = TRUE
            Rec_Cil_1_Gar_4 = FALSE

            Ava_Cil_1_Gar_5 = TRUE
            Rec_Cil_1_Gar_5 = FALSE

            Ava_Cil_1_Gar_6 = TRUE
            Rec_Cil_1_Gar_6 = FALSE

            Ava_Cil_2_Gar_1 = TRUE
            Rec_Cil_2_Gar_1 = FALSE

            Ava_Cil_2_Gar_2 = TRUE
            Rec_Cil_2_Gar_2 = FALSE

            Ava_Cil_2_Gar_3 = TRUE
            Rec_Cil_2_Gar_3 = FALSE

            Ava_Cil_2_Gar_4 = TRUE
            Rec_Cil_2_Gar_4 = FALSE

            Ava_Cil_2_Gar_5 = TRUE
            Rec_Cil_2_Gar_5 = FALSE

            Ava_Cil_2_Gar_6 = TRUE
            Rec_Cil_2_Gar_6 = FALSE


         CASE 181
            Abre_Gar_Triplo_Lado_A = TRUE
            Fecha_Gar_Triplo_Lado_A = FALSE

            Abre_Gar_Triplo_Lado_B = TRUE
            Fecha_Gar_Triplo_Lado_B = FALSE

            Abre_Comp_Indiv_Gar_1 = FALSE
            Fecha_Comp_Indiv_Gar_1 = TRUE

            Abre_Comp_Indiv_Gar_3 = FALSE
            Fecha_Comp_Indiv_Gar_3 = TRUE

            Abre_Comp_Indiv_Gar_4 = FALSE
            Fecha_Comp_Indiv_Gar_4 = TRUE

            Abre_Comp_Indiv_Gar_6 = FALSE
            Fecha_Comp_Indiv_Gar_6 = TRUE

            Ava_Cil_1_Gar_1 = TRUE
            Rec_Cil_1_Gar_1 = FALSE

            Ava_Cil_1_Gar_2 = TRUE
            Rec_Cil_1_Gar_2 = FALSE

            Ava_Cil_1_Gar_3 = TRUE
            Rec_Cil_1_Gar_3 = FALSE

            Ava_Cil_1_Gar_4 = TRUE
            Rec_Cil_1_Gar_4 = FALSE

            Ava_Cil_1_Gar_5 = TRUE
            Rec_Cil_1_Gar_5 = FALSE

            Ava_Cil_1_Gar_6 = TRUE
            Rec_Cil_1_Gar_6 = FALSE

            Ava_Cil_2_Gar_1 = TRUE
            Rec_Cil_2_Gar_1 = FALSE

            Ava_Cil_2_Gar_2 = TRUE
            Rec_Cil_2_Gar_2 = FALSE

            Ava_Cil_2_Gar_3 = TRUE
            Rec_Cil_2_Gar_3 = FALSE

            Ava_Cil_2_Gar_4 = TRUE
            Rec_Cil_2_Gar_4 = FALSE

            Ava_Cil_2_Gar_5 = TRUE
            Rec_Cil_2_Gar_5 = FALSE

            Ava_Cil_2_Gar_6 = TRUE
            Rec_Cil_2_Gar_6 = FALSE



      ENDSWITCH

end

--- ConfGarra.dat ---
&ACCESS RVO1
&PARAM EDITMASK = *
DEFDAT ConfGarra

ENDDAT
